{attribute 'qualified_only'}
{attribute 'strict'}
TYPE E_State :
(
	DISABLE		:= 0,
	READY 		:= 1,
	WARNING		:= 2,
	ERROR		:= 3
	
);
END_TYPE

(* stored: Version 1.1.0.1, ProductVersion 3.1.4024.12
   DUT E_State: Id {c83aa07a-7304-4757-afd4-52624ef9106d} *)
